(* CODESYS project MNG_SimIO.export

Project tree, tasks and I/O mapping:
  libraries: Standard, * (System); SysSocket, * (System); SysTypes, * (System); CmpErrors, * (System); CAA Callback Extern, * (CAA Technical Workgroup); SysMem, * (System); SysMem, * (System); CAA Callback Extern, * (CAA Technical Workgroup)
  task MNG_SIMIO (cyclic, interval 5 ms, priority 1) calls MNG_IO
  MNG_SimIO/
    data type MNG_DataArray
    data type MNG_DatagramHeader
    data type MNG_DatagramType
    data type MNG_RawDatagram
    data type POSE6
    data type TRAFO
    data type VEC3
    function CallbackReset [ST]
    function GetIPAddress [ST]
    program MNG_IO [ST]
    function block MNG_SIMIO_UPDATER [ST]
  data type MNG_APPLICATION_INPUTS_32BIT
  data type MNG_APPLICATION_OUTPUTS_32BIT
*)

// MNG_APPLICATION_INPUTS_32BIT
TYPE MNG_APPLICATION_INPUTS_32BIT :
STRUCT
    NumSignals                    : INT     := 5         ;
Drehschieber_Achse_1_RCHD: BOOL    := 0; (* STEP_Drehschieber_1_Drehschieber_Achse_1?KinReached *)

Drehschieber_Achse_1_AXIS: REAL    := 0.0; (* ng_STEP_Drehschieber_1_Drehschieber_Achse_1?KinAxis *)

Drehschieber_Achse_1_KinActPosOffset: REAL    := 0.0; (* Drehschieber_1_Drehschieber_Achse_1?KinActPosOffset *)

EndoflEnd_of_Line_Packaging_STEP_Set_AST_out: BOOL    := 0; (*  *)

EndoflEnd_of_Line_Packaging_STEP_Set_GST_out: BOOL    := 0; (*  *)

END_STRUCT
END_TYPE

// MNG_APPLICATION_OUTPUTS_32BIT
TYPE MNG_APPLICATION_OUTPUTS_32BIT :
STRUCT
    NumSignals                    : INT     := 3         ;
Drehschieber_Achse_1_TGT_POS: REAL    := 0.0; (*  *)

EndoflEnd_of_Line_Packaging_STEP_Ist_GST_out: BOOL    := 0; (* _EndoflEnd_of_Line_Packaging_STEP?Ist_GST_out *)

EndoflEnd_of_Line_Packaging_STEP_Ist_AST_out: BOOL    := 0; (* _EndoflEnd_of_Line_Packaging_STEP?Ist_AST_out *)

END_STRUCT
END_TYPE

// MNG_SimIO/MNG_DataArray
TYPE MNG_DataArray : ARRAY[1..1000] OF DWORD; END_TYPE

// MNG_SimIO/MNG_DatagramHeader
(* @END_DECLARATION := '0' *)
(* @NESTEDCOMMENTS := 'Yes' *)
(* @PATH := '\/MNG_SIMULATION' *)
(* @OBJECTFLAGS := '0, 8' *)
TYPE MNG_DatagramHeader :(* datagram header (4 byte aligned) *)
STRUCT
	(* Time when datagram has been created *)
	Counter 	: DWORD;
	(* Time when datagram has been sent *)
	SentTime 		: DWORD;
	(* Type of the datagram *)
	DatagramType 	: DWORD := MNG_DatagramType.MNG_UnknownDatagram;
	(* Byte count in the payload *)
	ByteCount 		: DWORD := 0;
END_STRUCT
END_TYPE

// MNG_SimIO/MNG_DatagramType
{attribute 'qualified_only'}
{attribute 'strict'}
TYPE MNG_DatagramType :
(
		(*Dead man datagram signalizing peer is alive *)
	MNG_DeadManDatagram := 0,
	(*Time tick synchonisation *)
	MNG_TimeTick,
	(*Time tick synchonisation *)
	MNG_TimeTickRequest,
	(*Initialization of the connection *)
	MNG_InitConnection,
	(*Reset simulation *)
	MNG_ResetSimulation,
	(*Rewind simulation *)
	MNG_RewindSimulation,
	(*Start simulation *)
	MNG_StartSimulation,
	(*Stop simulation *)
	MNG_StopSimulation,
	(*IO Config datagram *)
	MNG_IOConfig,
	(*Complete Raw IO Image *)
	MNG_RawIOImage,
	(*Complete Raw 32 Bit IO Image *)
	MNG_Raw32BitImage,
	(*Delta IO, only ios that have changed *)
	(* IODelta, *)
	(*Text datagram *)
	MNG_TextDatagram,
	(*Unknown Datagram (future updates of peer, not supported by this side) *)
	MNG_UnknownDatagram
);
END_TYPE

// MNG_SimIO/MNG_RawDatagram
(* @NESTEDCOMMENTS := 'Yes' *)
(* @PATH := '\/MNG_SIMULATION' *)
(* @OBJECTFLAGS := '0, 8' *)
TYPE MNG_RawDatagram :(* binary TCP/IP datagram (4 byte aligned) *)
STRUCT
	Header	:  MNG_DatagramHeader;(* datagram header *)
	Payload	:  MNG_DataARRAY;
END_STRUCT
END_TYPE

// MNG_SimIO/POSE6
(* @END_DECLARATION := '0' *)
(* @NESTEDCOMMENTS := 'Yes' *)
(* @PATH := '\/MNG_TCPIP' *)
TYPE POSE6 :(* position and orientation as an euler based pose *)
STRUCT
	x, y, z, a, b, c : REAL;
END_STRUCT
END_TYPE

// MNG_SimIO/TRAFO
(* @NESTEDCOMMENTS := 'Yes' *)
(* @PATH := '\/MNG_TCPIP' *)
TYPE TRAFO :(* position and orientation as a 4x4 matrix *)
STRUCT
	baseX : VEC3; 
	fill0 : REAL;
	baseY : VEC3; 
	fill1 : REAL;
	baseZ : VEC3; 
	fill2 : REAL;
	origin : VEC3;
	fill3 : REAL;
END_STRUCT
END_TYPE

// MNG_SimIO/VEC3
(* @END_DECLARATION := '0' *)
(* @NESTEDCOMMENTS := 'Yes' *)
(* @PATH := '\/MNG_TCPIP' *)
TYPE VEC3 :(* 3d position *)
STRUCT
	x, y, z : REAL;
END_STRUCT
END_TYPE

// MNG_SimIO/MNG_IO
PROGRAM MNG_IO
VAR_OUTPUT
        I : MNG_APPLICATION_INPUTS_32BIT;
END_VAR
VAR_INPUT
        Q : MNG_APPLICATION_OUTPUTS_32BIT;
END_VAR

VAR
	simIO : MNG_SIMIO_UPDATER;
END_VAR
(* @END_DECLARATION := '0' *)

simIO.Q := Q;
simIO(connect := TRUE);
I := simIO.I;

END_PROGRAM

// MNG_SimIO/MNG_SIMIO_UPDATER
FUNCTION_BLOCK MNG_SIMIO_UPDATER
(* This function block implements simple TCP/IP client protocol.              *)
(* The max. size of binary tx/rx data has to be <= PLCPRJ_BUFFER_SIZE         *)
VAR_INPUT
connect : BOOL := FALSE;
IPAddress : STRING := '192.168.8.175';
port : INT := 5004;
timeout : DINT := 3;		(* Timeout in seconds *)
Q : MNG_Application_Outputs_32Bit;    (* Tx user data *)
END_VAR
VAR_OUTPUT
I      : MNG_Application_Inputs_32Bit        ; (* Rx user data *)
Counter   : DINT := 0;
Connected : BOOL := FALSE;
END_VAR
VAR
state : INT := 0;
socket : RTS_IEC_HANDLE := -1(*SOCKET_INVALID*);
bOptNoDelay: BOOL := TRUE;
sa:SOCKADDRESS;
fdRead:SOCKET_FD_SET;
tvTimeout:SOCKET_TIMEVAL;
pdiReady:DINT := 0;
toServer         : MNG_RawDatagram;
fromServer       : MNG_RawDatagram;
expectedSize, recvSize : LINT := 0;
sendSize: UDINT := 0; 
sentSize : LINT := 0;

bInit: BOOL := FALSE;
DWordBuffer      : DWORD                                               ; (* convert DWORD data *)
DIntBuffer       : DINT                                                ; (* convert DINT data *)
Segment11_F: BOOL;
Error: DINT;
diSocket: BOOL;
result: RTS_IEC_RESULT; 
callback: CB.CB_CALLBACK;
callbackError: CB.ERROR; 
END_VAR
(* @END_DECLARATION := '0'                                                    *)

IF NOT bInit THEN
//         SysCallbackRegister(INDEXOF(CallbackReset), EVENT_BEFORE_RESET);
	callback.eEvent := CB.EVENT.BEFORE_RESET;
	callback.eClass := CB.EVENT_CLASS.ALL_CLASSES;
	callback.eSource := CB.EVENT_SOURCE.ALL_SOURCES;
	callback.pPOUFunc := ADR(CallbackReset); 
	
	CB.RegisterCallback(callback, ADR(callbackError));
        bInit := TRUE;
END_IF
CASE state OF
0:											(* Init *)
  	socket := -1(*SOCKET_INVALID*);
  	Connected := FALSE;
  	IF connect THEN
  	        state  := 10;
  	END_IF
10:											(* Create socket *)
        socket := SysSockCreate(SOCKET_AF_INET, SOCKET_STREAM, 0, ADR(result));
        (*IF socket <> 0(*= SOCKET_INVALID*) THEN
            state := 100;
        ELSE
            state := 20;
        END_IF*)
		state := 20;
20:											(* Setup and Connect *)
        (* SysSockSetOption(socket, SOCKET_SOL, SOCKET_SO_SNDBUF, ADR(diMaxDataSize), SIZEOF(diMaxDataSize));
        SysSockSetOption(socket, SOCKET_SOL, SOCKET_SO_RCVBUF, ADR(diMaxDataSize), SIZEOF(diMaxDataSize));
        lOptLinger.l_onoff:=0;
        lOptLinger.l_linger:=0;
        SysSockSetOption(diSocket,	SOCKET_SOL, SOCKET_SO_LINGER, ADR(lOptLinger), SIZEOF(lOptLinger)); *)
        bOptNoDelay:=TRUE;
        SysSockSetOption(socket,	SOCKET_IPPROTO_TCP, SOCKET_TCP_NODELAY, ADR(bOptNoDelay), SIZEOF(bOptNoDelay));
        sa.sin_family:=SOCKET_AF_INET;
        sa.sin_addr.ulAddr:=GetIPAddress(IPAddress);
        tvTimeout.tv_sec := timeout ;
        tvTimeout.tv_usec := 0;
        fdRead.fd_count := 1;
        fdRead.fd_array[0] := socket;
        IF sa.sin_addr.ulAddr = SOCKET_INADDR_NONE THEN
                state := 121;
        ELSE
                 sa.sin_port:=SysSockHtons(port);
                 IF SysSockConnect(socket, ADR(sa), SIZEOF(sa)) = 0  THEN
                        state := 30;
                 ELSE
                         Error := 10035(*SysSockGetLastErrorSync(socket)*);	
						(* Query reason why connect reported failure *)
                                         CASE  Error OF
                         10035: 			(* EWOULDBLOCK *)
                                 state := 30;
                         10056: 			 (* ALREADY_CONNECTED*)
                                 state := 30;
                         ELSE
                                 state := 60;
                         END_CASE
                END_IF
        END_IF
30:											(* Data exchange *)
                Connected := TRUE;
                fdRead.fd_array[0] := socket;
                IF (SysSockSelect(SOCKET_FD_SETSIZE, ADR(fdRead), 0, 0, ADR(tvTimeout), ADR(pdiReady)) = CmpErrors.Errors.ERR_OK) AND pdiReady > 0 THEN
                expectedSize := 16 + (I.NumSignals+1) * 4;
                recvSize := SysSockRecv(socket, ADR(fromServer), expectedSize, 0, ADR(result));
                IF result <> CmpErrors.Errors.ERR_OK OR expectedSize <= 0 THEN
                         state := 60;

                ELSIF expectedSize = recvSize THEN

                        (* correct header data *)
                        fromServer.Header.ByteCount   	 := SysSockNtohl(fromServer.Header.ByteCount);
                        Counter                        				:= SysSockNtohl(fromServer.Header.Counter);
                        fromServer.Header.SentTime  	   := SysSockNtohl(fromServer.Header.SentTime);
                        fromServer.Header.DatagramType := SysSockNtohl(fromServer.Header.DatagramType);

                        (* currently only use the data on a 32 Bit raw image *)
                        IF fromServer.Header.DatagramType = MNG_DatagramType.MNG_Raw32BitImage THEN
                                                        (* BOOL Drehschieber_Achse_1_RCHD *)
                                                        I.Drehschieber_Achse_1_RCHD := fromServer.Payload[2] <> 0;
                                                        (* REAL Drehschieber_Achse_1_AXIS *)
                                                        DWordBuffer := SysSockNtohl(fromServer.Payload[3]);
                                                        SysMemCpy(pDest := ADR(I.Drehschieber_Achse_1_AXIS), pSrc := ADR(DWordBuffer), udiCount := 4);
                                                        (* REAL Drehschieber_Achse_1_KinActPosOffset *)
                                                        DWordBuffer := SysSockNtohl(fromServer.Payload[4]);
                                                        SysMemCpy(pDest := ADR(I.Drehschieber_Achse_1_KinActPosOffset), pSrc := ADR(DWordBuffer), udiCount := 4);
                                                        (* BOOL EndoflEnd_of_Line_Packaging_STEP_Set_AST_out *)
                                                        I.EndoflEnd_of_Line_Packaging_STEP_Set_AST_out := fromServer.Payload[5] <> 0;
                                                        (* BOOL EndoflEnd_of_Line_Packaging_STEP_Set_GST_out *)
                                                        I.EndoflEnd_of_Line_Packaging_STEP_Set_GST_out := fromServer.Payload[6] <> 0;
                                        state :=  40;
                END_IF
                END_IF
                ELSE
                state := 60;
                END_IF
40:											(* Send data *)
        sendSize := 16 + (Q.NumSignals+1) * 4;
        (*IF (SysSockSelect(SOCKET_FD_SETSIZE, ADR(fdRead), 0, 0, ADR(tvTimeout), ADR(result)) > 0) THEN*)
          toServer.Header.ByteCount    := SysSockHtonl(sendSize-16);
          toServer.Header.DatagramType := SysSockHtonl(MNG_DatagramType.MNG_Raw32BitImage);
          toServer.Header.Counter      := SysSockHtonl(Counter);
          toServer.Payload[1] := SysSockHtonl(Q.NumSignals); (* number of signals *)
                                                        (* REAL Drehschieber_Achse_1_TGT_POS *)
                        SysMemCpy(pDest := ADR(DWordBuffer), pSrc := ADR(Q.Drehschieber_Achse_1_TGT_POS), udiCount := 4);
                        toServer.Payload[2] := SysSockHtonl(DWordBuffer);
                                                        (* BOOL EndoflEnd_of_Line_Packaging_STEP_Ist_GST_out *)
                        IF Q.EndoflEnd_of_Line_Packaging_STEP_Ist_GST_out = TRUE THEN
                            toServer.Payload[3] := 16#FFFFFFFF;   (*BOOL *)
                        ELSE
                            toServer.Payload[3] := 0;
                        END_IF;
                                                        (* BOOL EndoflEnd_of_Line_Packaging_STEP_Ist_AST_out *)
                        IF Q.EndoflEnd_of_Line_Packaging_STEP_Ist_AST_out = TRUE THEN
                            toServer.Payload[4] := 16#FFFFFFFF;   (*BOOL *)
                        ELSE
                            toServer.Payload[4] := 0;
                        END_IF;
        (*    toServer.Header.SentTime := SysSockHtonl(clock.systemTime.wMilliseconds + clock.systemTime.wMinute * 60000); *)
            sentSize := SysSockSend(socket, ADR(toServer), sendSize, 0, ADR(result));
            IF sentSize < 0 THEN
               state := 60;
            ELSE
               state := 30;
            END_IF
        (*ELSE
                        state := 60;
        END_IF*)
60:											(* Disconnect *)
                IF socket = 0(*SOCKET_INVALID*) THEN
                                state := 0;
                ELSE
                                IF SysSockClose(socket) <> 0(*= FALSE*) THEN
                                          state := 161;
                                ELSE
                                                state := 70;
                                END_IF
          END_IF
70:											(* Delete socket *)
          IF socket = 0(*SOCKET_INVALID*) THEN
                                state := 0;
                ELSE
                    IF SysSockShutdown(socket, 0) <> 0(*= FALSE*) THEN
                                          state := 0;
                                ELSE
                                                state := 0;
                                END_IF
          END_IF
110:										(* Error Create socket failed *)
;
121:										(* Error IP number invalid *)
;
122:										(* Error connect failed *)
     state := 70;
131:										(* Error while receiving, received bytes < expected)*)
                 state := 60;
161: 										(* Error close failed *)
;
END_CASE
IF NOT connect AND state> 0 AND state < 60 THEN
                state := 60;
END_IF

END_FUNCTION_BLOCK

// MNG_SimIO/CallbackReset
FUNCTION CallbackReset : BOOL
VAR_INPUT
	dwSpec  : DWORD; (* CB.Event and CB.EventClass *)
	 dwParam : DWORD; (* Application specific Parameter *)
	 dwSource : DWORD; (* CB.EventSource *)
END_VAR
VAR
END_VAR

IF CB.DecodeEvent(dwSpec) = CB.EVENT.BEFORE_RESET THEN
    IF MNG_IO.simIO.socket <> -1 THEN
		SysSockClose(MNG_IO.simIO.socket);
	END_IF
END_IF

END_FUNCTION

// MNG_SimIO/GetIPAddress
FUNCTION GetIPAddress : UDINT
VAR_INPUT
	stIPAddress:STRING;		(* IP-address or computer name *)
END_VAR
VAR
	diIPAddress:UDINT := SOCKET_INADDR_NONE;
END_VAR

SysSockInetAddr(stIPAddress, ADR(diIPAddress));
IF diIPAddress = SOCKET_INADDR_NONE THEN
	SysSockGetHostByName(stIPAddress, ADR(diIPAddress));
END_IF
GetIPAddress:=diIPAddress;

END_FUNCTION
